TYPE ST_MotionlinxAI_Controller_Config :
	STRUCT
		ExtendTime	: LREAL;
		RetractTime : LREAL;
	END_STRUCT
END_TYPE

(* stored: Version 1.1.0.1, ProductVersion 3.1.4024.15
   DUT ST_MotionlinxAI_Controller_Config: Id {2b2e9d12-22c7-4af5-b0ca-309c13117547} *)
